PROGRAM AxisAction
VAR
	bBoot : BOOL := true;

	bMove: BOOL;
	tof_PowerOff: TOF;
	ldf_PowerOff: F_TRIG;
END_VAR

IF bBoot THEN
	initAction();
	bBoot := FALSE;
END_IF



Axis.FeedCar();

METHOD initAction : BOOL
VAR_INPUT
END_VAR
FeedCar.Encoder := ADR(axis.FeedCar_Enc);

FeedCar.Set_VFD_IO(
	FWD:= ADR(io.q104), 
	REV:= ADR(io.q105), 
	Speed_Io_1:= ADR(io.q106), 
	Speed_Io_2:= ADR(io.q107), 
	Speed_Io_3:= ADR(io.q108), 
	Reset:= ADR(io.q307), 
	Run:= ADR(io.i107), 
	Error:= ADR(io.i108)
);

FeedCar.SetLimit_IO(
	Origin:= ADR(io.i213), 
	P_Limit:= 0, 
	N_Limit:= 0
);

FeedCar.Name := "FeedCar";
END_METHOD

END_PROGRAM

(* stored: Version 1.1.0.1, ProductVersion 3.1.4024.15
   POU AxisAction: Id {d2c76a6c-08c2-4d2b-84d6-d1bbec5e06db}, SpecialFunc None
   Method initAction: Id {807103db-1c2a-4b9a-b1e6-e9fe86703db7} *)
